ABB RAPID module: Comunicacao

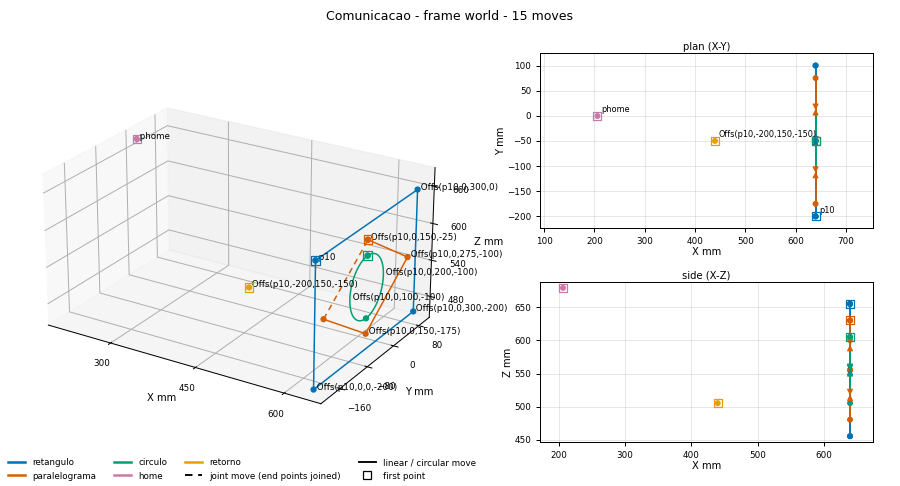
[picture p0: tool path of Comunicacao in frame world, 15 of 15 moves have a stored position in this frame; points joined in program order, loops and branches not executed]
MODULE Module1
    CONST robtarget p10:=[[639.86,-200.00,655.30],[0.500001,3.77523E-06,0.866025,-8.30828E-06],[-1,0,-1,0],[9E+09,9E+09,9E+09,9E+09,9E+09,9E+09]];
    CONST robtarget phome:=[[205.97,-0.43,679.40],[0.500002,-1.72274E-06,0.866024,-2.13775E-07],[-1,0,-1,0],[9E+09,9E+09,9E+09,9E+09,9E+09,9E+09]];
    PROC main()
        TPErase;
        TPReadFK reg1, "Bom dia meu lindo, escolha uma das opções", stEmpty, "RETANGULO", "PARALELOGRAMA", "CIRCULO", "BANDEIRA";
        !Inicio
        home;
        retorno;
        !Condição
        IF reg1=2 THEN
            retangulo;
        ELSEIF reg1=3 THEN
            paralelograma;
        ELSEIF reg1=4 THEN
            circulo;
        ELSEIF reg1=5 THEN
            bandeira;
        ENDIF
        !Final
        retorno;
        home;
        TPErase;
        TPReadFK reg2, "A ROTINA FOI EXECUTADA CORRETAMENTE?", stEmpty, "SIM", stEmpty, "NAO", stEmpty;
        IF reg2=4 THEN
            main;
        ENDIF
    ENDPROC

    PROC retangulo()
        MoveJ p10, vmax, fine, tool0;
        MoveL Offs(p10, 0, 300, 0), vmax, fine, tool0;
        MoveL Offs(p10, 0, 300, -200), vmax, fine, tool0;
        MoveL Offs(p10, 0, 0, -200), vmax, fine, tool0;
        MoveL p10, vmax, fine, tool0;
    ENDPROC
    PROC paralelograma()
        MoveJ Offs(p10, 0, 150, -25), vmax, fine, tool0;
        MoveL Offs(p10, 0, 275, -100), vmax, fine, tool0;
        MoveL Offs(p10, 0, 150, -175), vmax, fine, tool0;
        MoveL Offs(p10, 0, 25, -100), vmax, fine, tool0;
        MoveJ Offs(p10, 0, 150, -25), vmax, fine, tool0;
    ENDPROC
    PROC circulo()
        MoveJ Offs(p10, 0, 150, -50), vmax, fine, tool0;
        MoveC Offs(p10, 0, 200, -100), Offs(p10, 0, 150, -150), vmax, fine, tool0;
        MoveC Offs(p10, 0, 100, -100), Offs(p10, 0, 150, -50), vmax, fine, tool0;
    ENDPROC
    PROC bandeira()
        retangulo;
        retorno;
        paralelograma;
        retorno;
        circulo;
    ENDPROC
    PROC home()
        MoveJ phome, vmax, fine, tool0;
    ENDPROC
    PROC retorno()
        MoveJ Offs(p10, -200, 150, -150), vmax, fine, tool0;
    ENDPROC
ENDMODULE
